{attribute 'qualified_only'}
{attribute 'strict'}
{attribute 'to_string'}
TYPE CdEventSeverity :
(
    Verbose:=0,     // Useful Information for debugging 
    Info:=1,        // Useful Information for operators
    Warning:=2,     // Machine operation not inhibited but at risk of becoming so
    Error:=3,       // Component operation blocked till resolved
    Critical:=4,    // Machine operation bloced till resolved
	                // 5-7 Reserved for future implementaion
	Lockout:=8      // Mackine locked out from use until ADMIN clears Fault 
					// 9 Reserved for future implementaion 
	
);
END_TYPE

(* stored: Version 1.1.0.1, ProductVersion 3.1.4024.15
   EnumerationTextList CdEventSeverity: Id {35d3193d-3c8b-4104-8260-5814f9cf34bf} *)
